// Communicates with the TraceTek hardware over Modbus to get more information about a leak
FUNCTION_BLOCK FB_TraceTekModbus
VAR_INPUT
	nModbusSlaveAddress : BYTE; // Modbus address of slave to be read from
	bLeakDetected : BOOL; // Whether a leak has been detected
	bResetError : BOOL; // Reset signal for error
END_VAR
VAR_OUTPUT
	{attribute 'pytmc' := '
		pv: LOC_RES
		io: input
	'}
	nLocationResistance: UINT; // Used for calculating the location of the leak
	{attribute 'pytmc' := '
		pv: ERROR
		io: i
		field: OSV MAJOR
		field: ZSV NO_ALARM
		field: ZNAM OK
		field: ONAM ERROR
	'}
	bError : BOOL := FALSE; // Flag for Modbus communication errors
	nErrorId : MODBUS_ERRORS := MODBUS_ERRORS.MODBUSERROR_NO_ERROR; // Description of Modbus error
END_VAR
VAR
	aModbusBuffer : WORD := 16#FFFF;  // Infinite until real value is read from device
	fbModbusMaster : ModbusRtuMaster_KL6x22B := (
		Quantity := 1,
		MBAddr := 1,
		cbLength := SIZEOF(aModbusBuffer),
		pMemoryAddr := ADR(aModbusBuffer),
		Timeout := T#5S
	);
END_VAR

IF bResetError THEN // Reset modbus error
	bError := FALSE;
	nErrorId := MODBUS_ERRORS.MODBUSERROR_NO_ERROR;
END_IF

// Update modbus status
fbModbusMaster.Execute := FALSE;
fbModbusMaster.ReadInputRegs();

IF fbModbusMaster.Error THEN
	bError := TRUE;
	nErrorId := fbModbusMaster.ErrorId;
END_IF

IF NOT fbModbusMaster.BUSY AND bLeakDetected THEN // Start reading
	fbModbusMaster.UnitID := nModbusSlaveAddress;
	fbModbusMaster.Execute := TRUE;
	fbModbusMaster.ReadInputRegs();
END_IF

nLocationResistance := WORD_TO_UINT(aModbusBuffer);

END_FUNCTION_BLOCK

(* stored: Version 1.1.0.1, ProductVersion 3.1.4020.14
   POU FB_TraceTekModbus: Id {0f7af4f5-240b-40c0-81d3-4ad14d941ee4}, SpecialFunc None *)
